{attribute 'qualified_only'}
{attribute 'strict'}
TYPE E_SocketReceiveState :
(
	READY,
	RECEIVING,
	DONE,
	ERROR
);
END_TYPE

(* stored: Version 1.1.0.1, ProductVersion 3.1.4024.13
   DUT E_SocketReceiveState: Id {0f493829-dece-4b66-88f8-8fce4b87752a} *)
